// TIA Portal V19 export
TYPE "UDT_DELAYON"
   STRUCT
      in : Struct
         spon { S7_SetPoint := 'True'} : Real := 0.0;   // Setpoint for delay on timer (Real number because we count every 100ms)
      END_STRUCT;
      don : Struct
         trigger : Bool := false;
         sp : Int := 0;
         actual : Int := 0;
         end : Bool := false;
      END_STRUCT;
      out : Struct
         on : Bool := false;
      END_STRUCT;
   END_STRUCT;
END_TYPE
